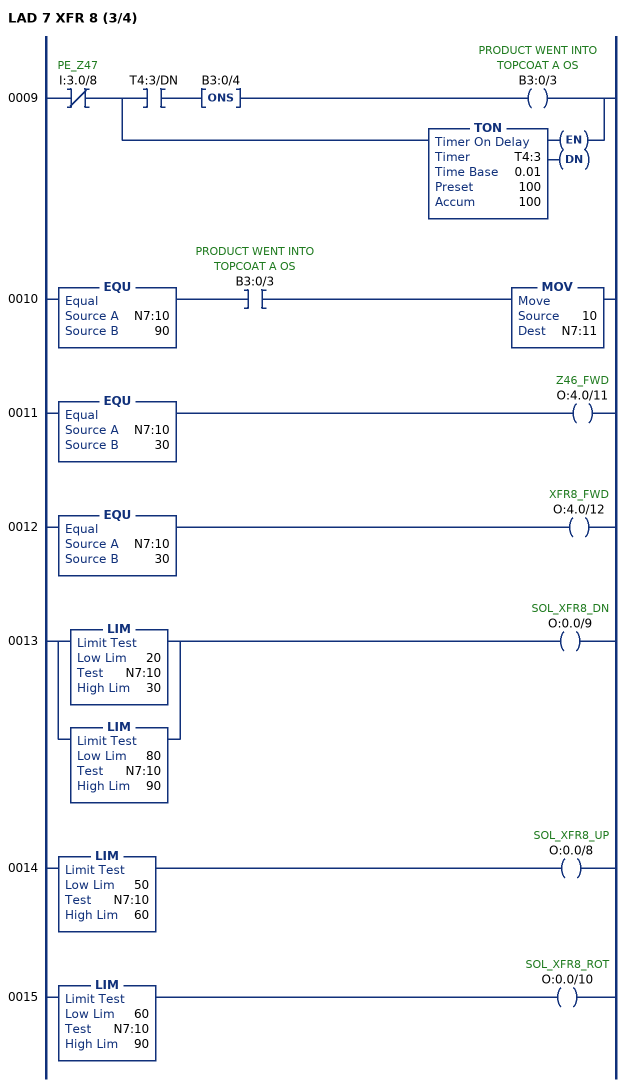
% Rung: 9 %
SOR XIO I:3.0/8 BST XIC T4:3/DN ONS B3:0/4 OTE B3:0/3 NXB TON T4:3 0.01 100 100 BND EOR
%   I:3.0/8  PE_Z47 %
%   B3:0/3  "PRODUCT WENT INTO TOPCOAT A OS" %
% Rung: 10 %
SOR EQU N7:10 90 XIC B3:0/3 MOV 10 N7:11 EOR
%   B3:0/3  "PRODUCT WENT INTO TOPCOAT A OS" %
% Rung: 11 %
SOR EQU N7:10 30 OTE O:4.0/11 EOR
%   O:4.0/11  Z46_FWD %
% Rung: 12 %
SOR EQU N7:10 30 OTE O:4.0/12 EOR
%   O:4.0/12  XFR8_FWD %
% Rung: 13 %
SOR BST LIM 20 N7:10 30 NXB LIM 80 N7:10 90 BND OTE O:0.0/9 EOR
%   O:0.0/9  SOL_XFR8_DN %
% Rung: 14 %
SOR LIM 50 N7:10 60 OTE O:0.0/8 EOR
%   O:0.0/8  SOL_XFR8_UP %
% Rung: 15 %
SOR LIM 60 N7:10 90 OTE O:0.0/10 EOR
%   O:0.0/10  SOL_XFR8_ROT %

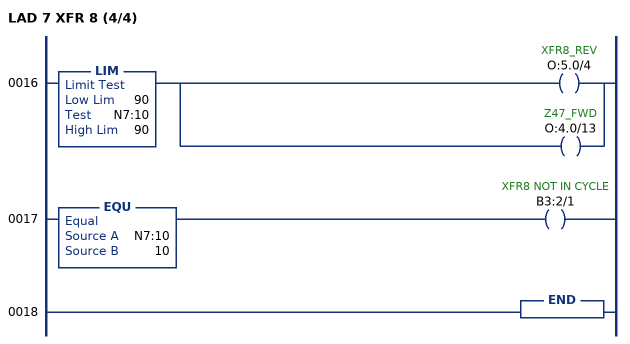
% Rung: 16 %
SOR LIM 90 N7:10 90 BST OTE O:5.0/4 NXB OTE O:4.0/13 BND EOR
%   O:5.0/4  XFR8_REV %
%   O:4.0/13  Z47_FWD %
% Rung: 17 %
SOR EQU N7:10 10 OTE B3:2/1 EOR
%   B3:2/1  "XFR8 NOT IN CYCLE" %
% Rung: 18 %
SOR END EOR

LADDER 8 "XFR 9"
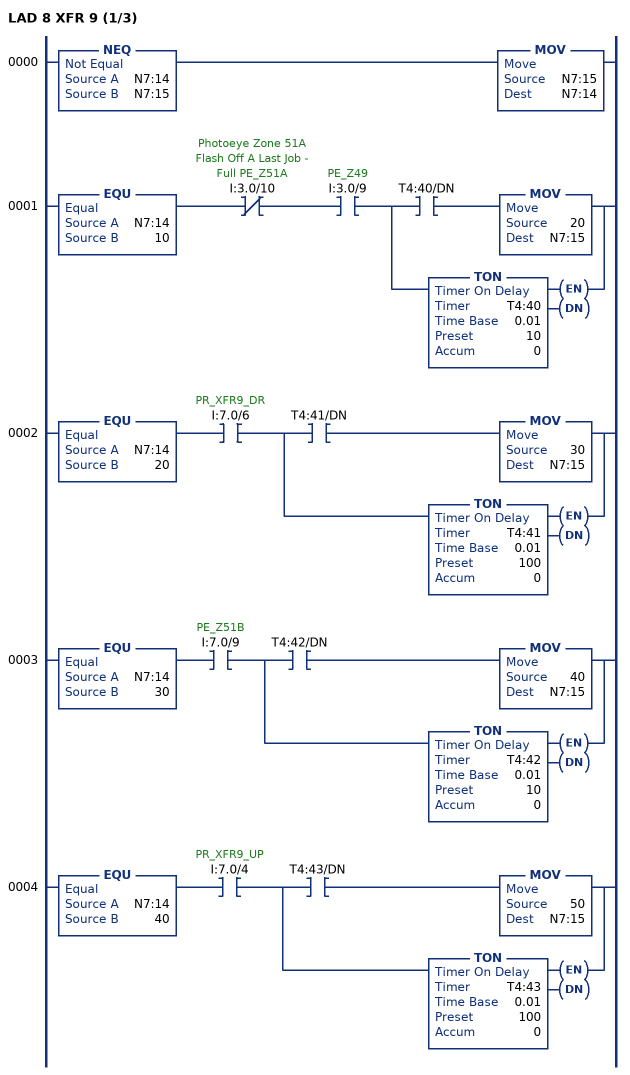
% Rung: 0 %
SOR NEQ N7:14 N7:15 MOV N7:15 N7:14 EOR
% Rung: 1 %
SOR EQU N7:14 10 XIO I:3.0/10 XIC I:3.0/9 BST XIC T4:40/DN MOV 20 N7:15 NXB TON T4:40 0.01 10 0 BND EOR
%   I:3.0/10  PE_Z51A  "Photoeye Zone 51A Flash Off A Last Job - Full" %
%   I:3.0/9  PE_Z49 %
% Rung: 2 %
SOR EQU N7:14 20 XIC I:7.0/6 BST XIC T4:41/DN MOV 30 N7:15 NXB TON T4:41 0.01 100 0 BND EOR
%   I:7.0/6  PR_XFR9_DR %
% Rung: 3 %
SOR EQU N7:14 30 XIC I:7.0/9 BST XIC T4:42/DN MOV 40 N7:15 NXB TON T4:42 0.01 10 0 BND EOR
%   I:7.0/9  PE_Z51B %
% Rung: 4 %
SOR EQU N7:14 40 XIC I:7.0/4 BST XIC T4:43/DN MOV 50 N7:15 NXB TON T4:43 0.01 100 0 BND EOR
%   I:7.0/4  PR_XFR9_UP %

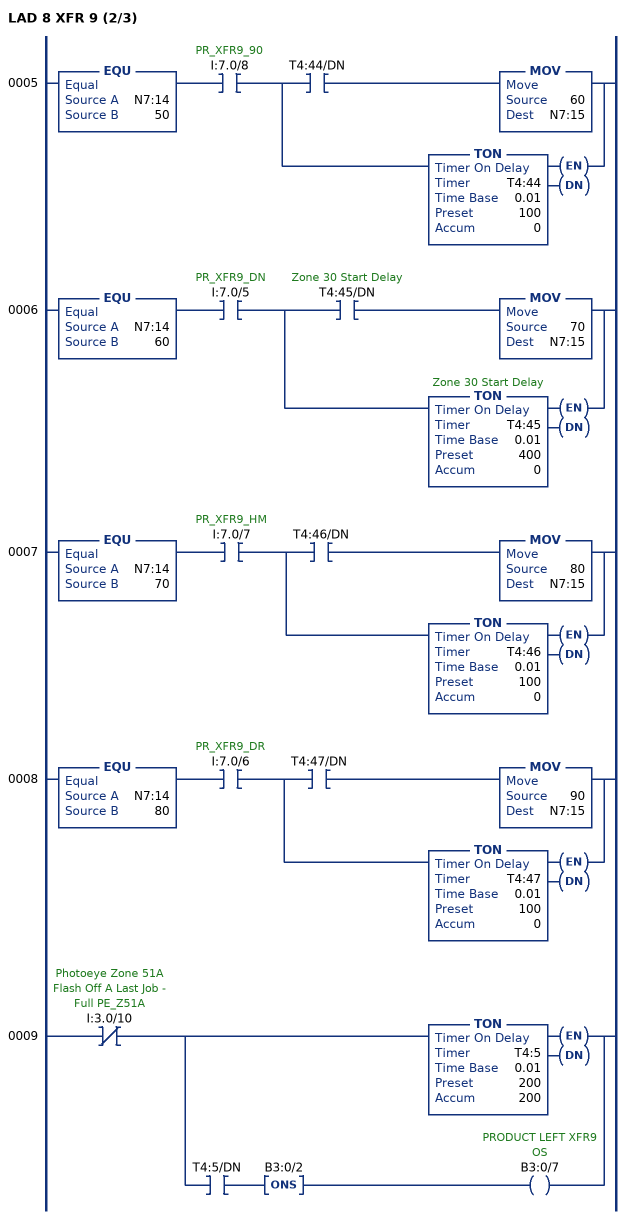
% Rung: 5 %
SOR EQU N7:14 50 XIC I:7.0/8 BST XIC T4:44/DN MOV 60 N7:15 NXB TON T4:44 0.01 100 0 BND EOR
%   I:7.0/8  PR_XFR9_90 %
% Rung: 6 %
SOR EQU N7:14 60 XIC I:7.0/5 BST XIC T4:45/DN MOV 70 N7:15 NXB TON T4:45 0.01 400 0 BND EOR
%   I:7.0/5  PR_XFR9_DN %
%   T4:45  "Zone 30 Start Delay" %
% Rung: 7 %
SOR EQU N7:14 70 XIC I:7.0/7 BST XIC T4:46/DN MOV 80 N7:15 NXB TON T4:46 0.01 100 0 BND EOR
%   I:7.0/7  PR_XFR9_HM %
% Rung: 8 %
SOR EQU N7:14 80 XIC I:7.0/6 BST XIC T4:47/DN MOV 90 N7:15 NXB TON T4:47 0.01 100 0 BND EOR
%   I:7.0/6  PR_XFR9_DR %
% Rung: 9 %
SOR XIO I:3.0/10 BST TON T4:5 0.01 200 200 NXB XIC T4:5/DN ONS B3:0/2 OTE B3:0/7 BND EOR
%   I:3.0/10  PE_Z51A  "Photoeye Zone 51A Flash Off A Last Job - Full" %
%   B3:0/7  "PRODUCT LEFT XFR9 OS" %

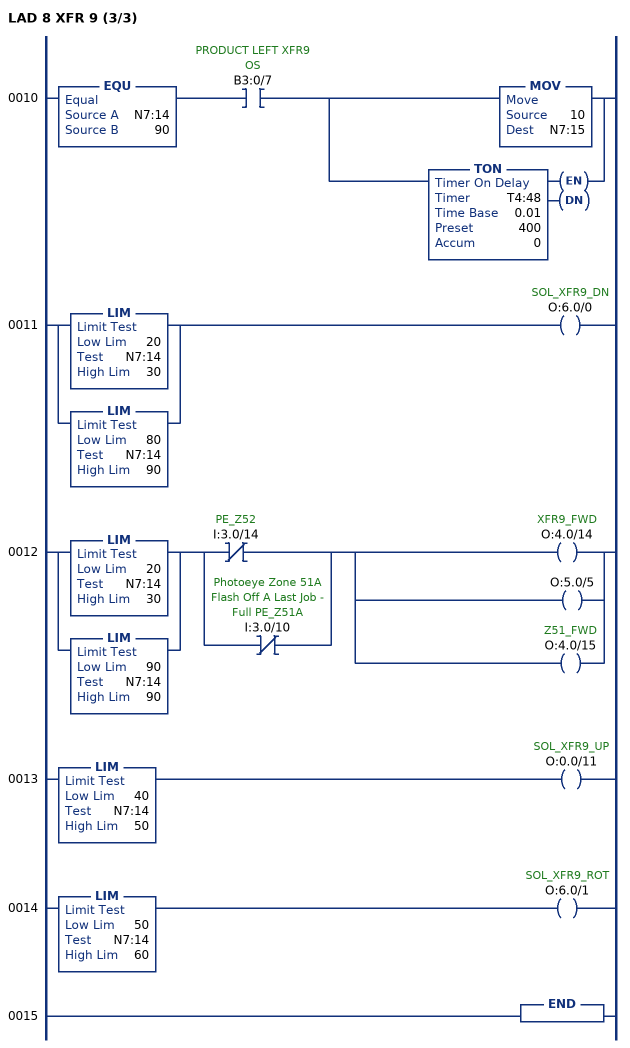
% Rung: 10 %
SOR EQU N7:14 90 XIC B3:0/7 BST MOV 10 N7:15 NXB TON T4:48 0.01 400 0 BND EOR
%   B3:0/7  "PRODUCT LEFT XFR9 OS" %
% Rung: 11 %
SOR BST LIM 20 N7:14 30 NXB LIM 80 N7:14 90 BND OTE O:6.0/0 EOR
%   O:6.0/0  SOL_XFR9_DN %
% Rung: 12 %
SOR BST LIM 20 N7:14 30 NXB LIM 90 N7:14 90 BND BST XIO I:3.0/14 NXB XIO I:3.0/10 BND BST OTE O:4.0/14 NXB OTE O:5.0/5 NXB OTE O:4.0/15 BND EOR
%   I:3.0/14  PE_Z52 %
%   I:3.0/10  PE_Z51A  "Photoeye Zone 51A Flash Off A Last Job - Full" %
%   O:4.0/14  XFR9_FWD %
%   O:4.0/15  Z51_FWD %
% Rung: 13 %
SOR LIM 40 N7:14 50 OTE O:0.0/11 EOR
%   O:0.0/11  SOL_XFR9_UP %
% Rung: 14 %
SOR LIM 50 N7:14 60 OTE O:6.0/1 EOR
%   O:6.0/1  SOL_XFR9_ROT %
% Rung: 15 %
SOR END EOR

LADDER 9 "XFR 10"
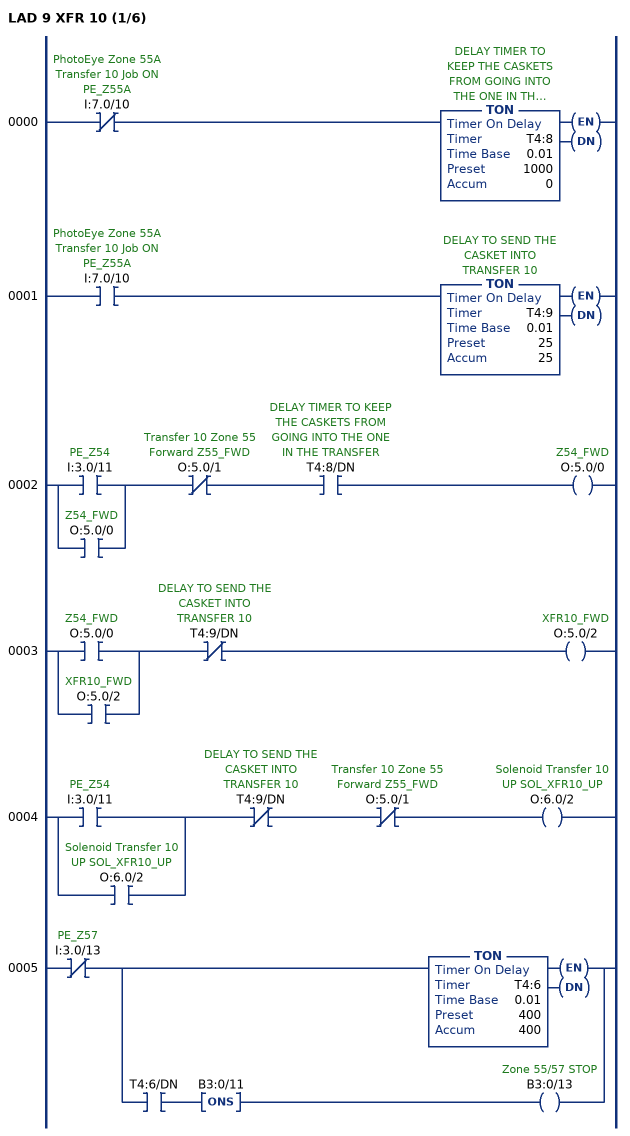
% Rung: 0 %
SOR XIO I:7.0/10 TON T4:8 0.01 1000 0 EOR
%   I:7.0/10  PE_Z55A  "PhotoEye Zone 55A Transfer 10 Job ON" %
%   T4:8  "DELAY TIMER TO KEEP THE CASKETS FROM GOING INTO THE ONE IN THE TRANSFER" %
% Rung: 1 %
SOR XIC I:7.0/10 TON T4:9 0.01 25 25 EOR
%   I:7.0/10  PE_Z55A  "PhotoEye Zone 55A Transfer 10 Job ON" %
%   T4:9  "DELAY TO SEND THE CASKET INTO TRANSFER 10" %
% Rung: 2 %
SOR BST XIC I:3.0/11 NXB XIC O:5.0/0 BND XIO O:5.0/1 XIC T4:8/DN OTE O:5.0/0 EOR
%   I:3.0/11  PE_Z54 %
%   O:5.0/0  Z54_FWD %
%   O:5.0/1  Z55_FWD  "Transfer 10 Zone 55 Forward" %
%   T4:8  "DELAY TIMER TO KEEP THE CASKETS FROM GOING INTO THE ONE IN THE TRANSFER" %
% Rung: 3 %
SOR BST XIC O:5.0/0 NXB XIC O:5.0/2 BND XIO T4:9/DN OTE O:5.0/2 EOR
%   O:5.0/0  Z54_FWD %
%   O:5.0/2  XFR10_FWD %
%   T4:9  "DELAY TO SEND THE CASKET INTO TRANSFER 10" %
% Rung: 4 %
SOR BST XIC I:3.0/11 NXB XIC O:6.0/2 BND XIO T4:9/DN XIO O:5.0/1 OTE O:6.0/2 EOR
%   I:3.0/11  PE_Z54 %
%   O:6.0/2  SOL_XFR10_UP  "Solenoid Transfer 10 UP" %
%   T4:9  "DELAY TO SEND THE CASKET INTO TRANSFER 10" %
%   O:5.0/1  Z55_FWD  "Transfer 10 Zone 55 Forward" %
% Rung: 5 %
SOR XIO I:3.0/13 BST TON T4:6 0.01 400 400 NXB XIC T4:6/DN ONS B3:0/11 OTE B3:0/13 BND EOR
%   I:3.0/13  PE_Z57 %
%   B3:0/13  "Zone 55/57 STOP" %

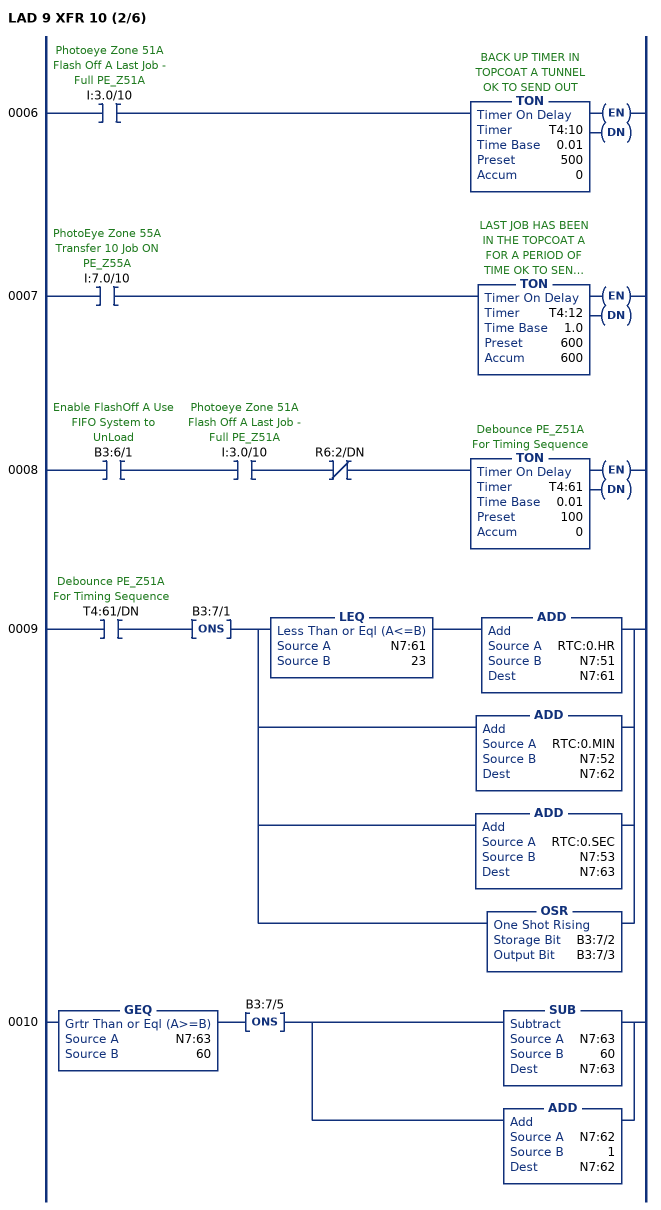
% Rung: 6 %
SOR XIC I:3.0/10 TON T4:10 0.01 500 0 EOR
%   I:3.0/10  PE_Z51A  "Photoeye Zone 51A Flash Off A Last Job - Full" %
%   T4:10  "BACK UP TIMER IN TOPCOAT A TUNNEL OK TO SEND OUT" %
% Rung: 7 %
SOR XIC I:7.0/10 TON T4:12 1.0 600 600 EOR
%   I:7.0/10  PE_Z55A  "PhotoEye Zone 55A Transfer 10 Job ON" %
%   T4:12  "LAST JOB HAS BEEN IN THE TOPCOAT A FOR A PERIOD OF TIME OK TO SEND OUT" %
% Rung: 8 %
SOR XIC B3:6/1 XIC I:3.0/10 XIO R6:2/DN TON T4:61 0.01 100 0 EOR
%   B3:6/1  "Enable FlashOff A Use FIFO System to UnLoad" %
%   I:3.0/10  PE_Z51A  "Photoeye Zone 51A Flash Off A Last Job - Full" %
%   T4:61  "Debounce PE_Z51A For Timing Sequence" %
% Rung: 9 %
SOR XIC T4:61/DN ONS B3:7/1 BST LEQ N7:61 23 ADD RTC:0.HR N7:51 N7:61 NXB ADD RTC:0.MIN N7:52 N7:62 NXB ADD RTC:0.SEC N7:53 N7:63 NXB OSR B3:7/2 B3:7/3 BND EOR
%   T4:61  "Debounce PE_Z51A For Timing Sequence" %
%   B3:7/3  "One Shot Rising FlashOff A Load Time into Stack" %
% Rung: 10 %
SOR GEQ N7:63 60 ONS B3:7/5 BST SUB N7:63 60 N7:63 NXB ADD N7:62 1 N7:62 BND EOR

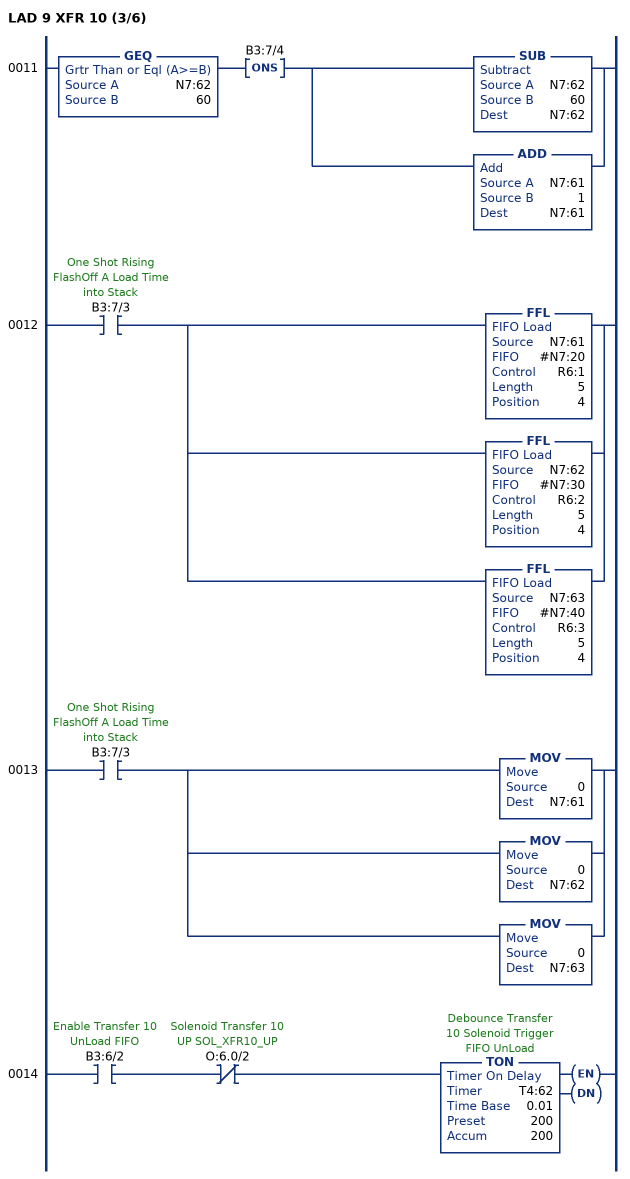
% Rung: 11 %
SOR GEQ N7:62 60 ONS B3:7/4 BST SUB N7:62 60 N7:62 NXB ADD N7:61 1 N7:61 BND EOR
% Rung: 12 %
SOR XIC B3:7/3 BST FFL N7:61 #N7:20 R6:1 5 4 NXB FFL N7:62 #N7:30 R6:2 5 4 NXB FFL N7:63 #N7:40 R6:3 5 4 BND EOR
%   B3:7/3  "One Shot Rising FlashOff A Load Time into Stack" %
% Rung: 13 %
SOR XIC B3:7/3 BST MOV 0 N7:61 NXB MOV 0 N7:62 NXB MOV 0 N7:63 BND EOR
%   B3:7/3  "One Shot Rising FlashOff A Load Time into Stack" %
% Rung: 14 %
SOR XIC B3:6/2 XIO O:6.0/2 TON T4:62 0.01 200 200 EOR
%   B3:6/2  "Enable Transfer 10 UnLoad FIFO" %
%   O:6.0/2  SOL_XFR10_UP  "Solenoid Transfer 10 UP" %
%   T4:62  "Debounce Transfer 10 Solenoid Trigger FIFO UnLoad" %

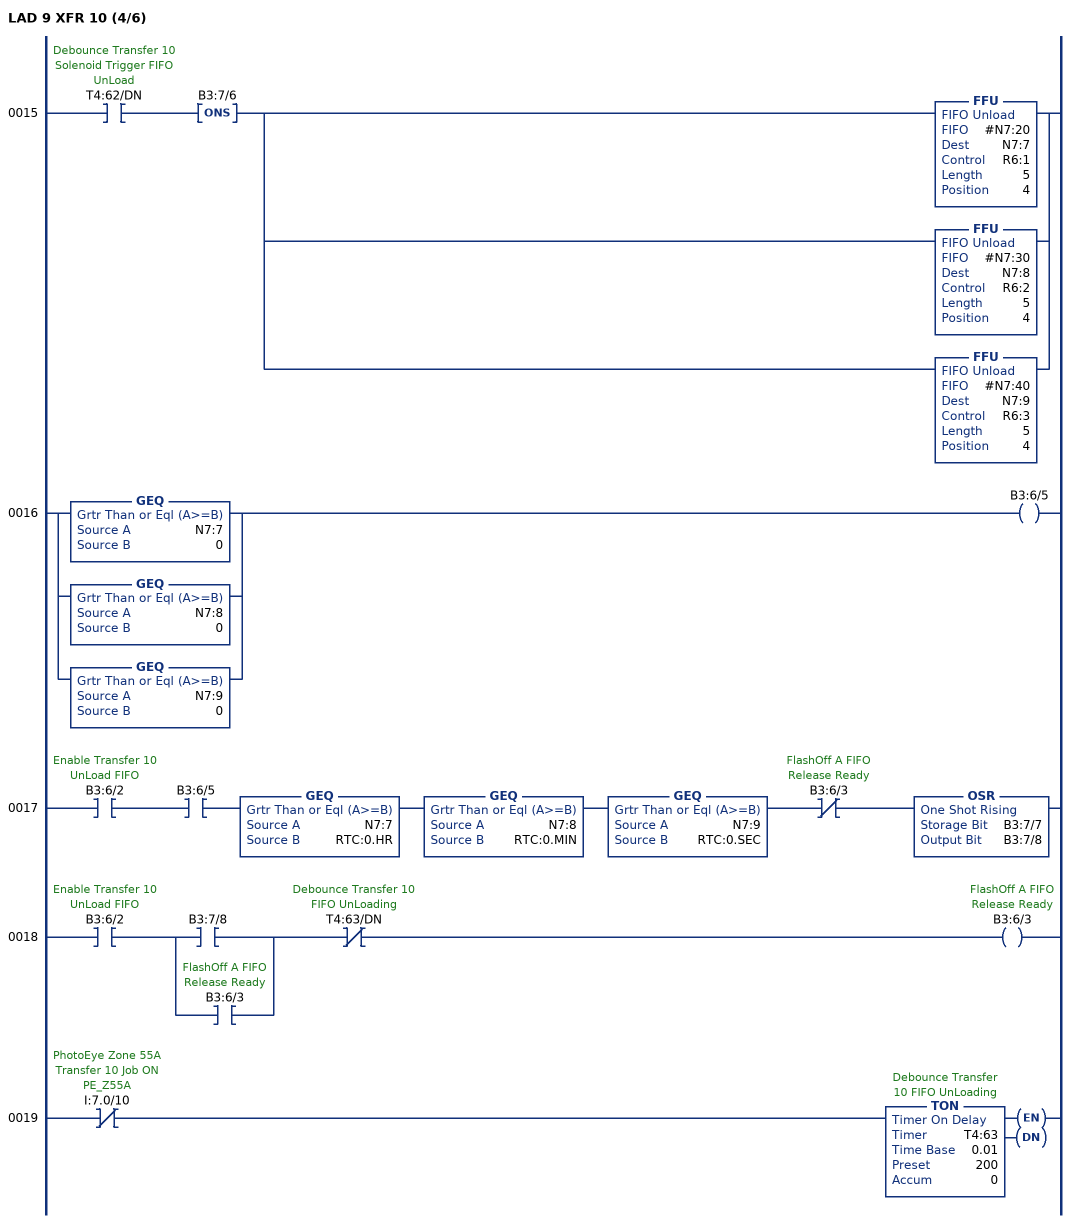
% Rung: 15 %
SOR XIC T4:62/DN ONS B3:7/6 BST FFU #N7:20 N7:7 R6:1 5 4 NXB FFU #N7:30 N7:8 R6:2 5 4 NXB FFU #N7:40 N7:9 R6:3 5 4 BND EOR
%   T4:62  "Debounce Transfer 10 Solenoid Trigger FIFO UnLoad" %
% Rung: 16 %
SOR BST GEQ N7:7 0 NXB GEQ N7:8 0 NXB GEQ N7:9 0 BND OTE B3:6/5 EOR
% Rung: 17 %
SOR XIC B3:6/2 XIC B3:6/5 GEQ N7:7 RTC:0.HR GEQ N7:8 RTC:0.MIN GEQ N7:9 RTC:0.SEC XIO B3:6/3 OSR B3:7/7 B3:7/8 EOR
%   B3:6/2  "Enable Transfer 10 UnLoad FIFO" %
%   B3:6/3  "FlashOff A FIFO Release Ready" %
% Rung: 18 %
SOR XIC B3:6/2 BST XIC B3:7/8 NXB XIC B3:6/3 BND XIO T4:63/DN OTE B3:6/3 EOR
%   B3:6/2  "Enable Transfer 10 UnLoad FIFO" %
%   B3:6/3  "FlashOff A FIFO Release Ready" %
%   T4:63  "Debounce Transfer 10 FIFO UnLoading" %
% Rung: 19 %
SOR XIO I:7.0/10 TON T4:63 0.01 200 0 EOR
%   I:7.0/10  PE_Z55A  "PhotoEye Zone 55A Transfer 10 Job ON" %
%   T4:63  "Debounce Transfer 10 FIFO UnLoading" %

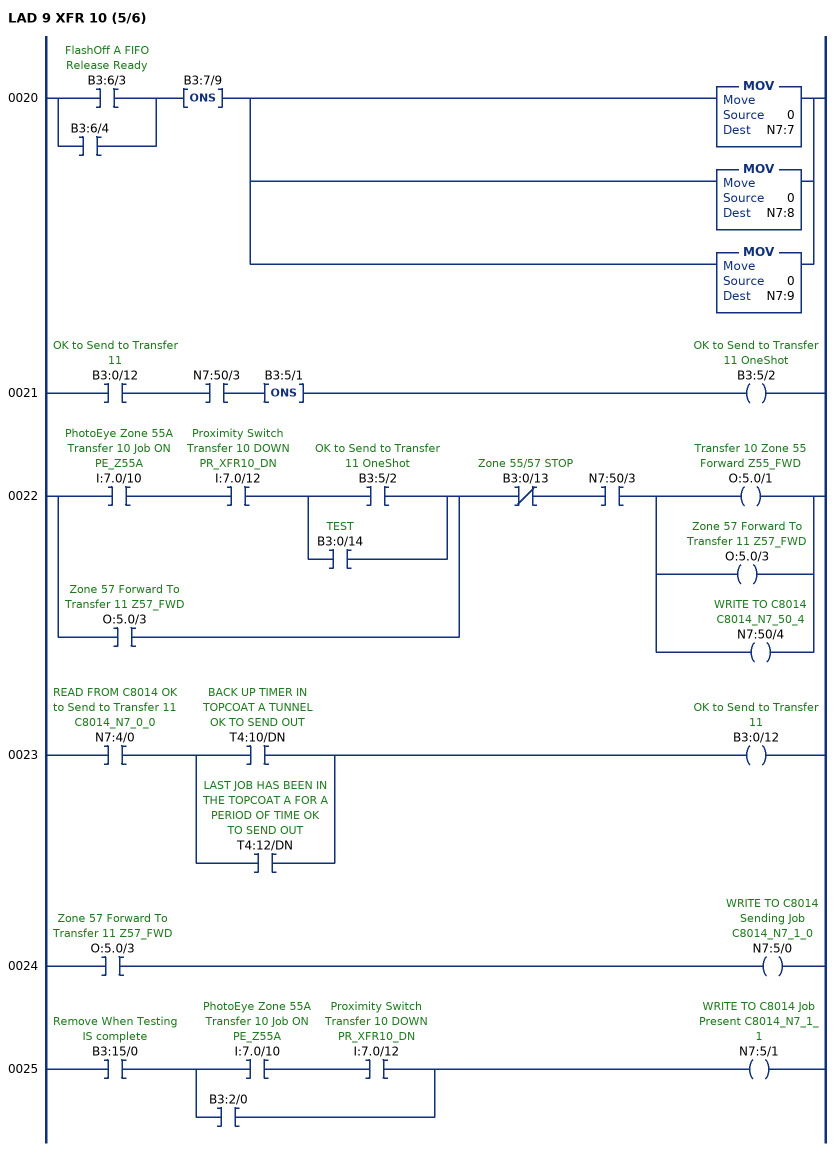
% Rung: 20 %
SOR BST XIC B3:6/3 NXB XIC B3:6/4 BND ONS B3:7/9 BST MOV 0 N7:7 NXB MOV 0 N7:8 NXB MOV 0 N7:9 BND EOR
%   B3:6/3  "FlashOff A FIFO Release Ready" %
% Rung: 21 %
SOR XIC B3:0/12 XIC N7:50/3 ONS B3:5/1 OTE B3:5/2 EOR
%   B3:0/12  "OK to Send to Transfer 11" %
%   B3:5/2  "OK to Send to Transfer 11 OneShot" %
% Rung: 22 %
SOR BST XIC I:7.0/10 XIC I:7.0/12 BST XIC B3:5/2 NXB XIC B3:0/14 BND NXB XIC O:5.0/3 BND XIO B3:0/13 XIC N7:50/3 BST OTE O:5.0/1 NXB OTE O:5.0/3 NXB OTE N7:50/4 BND EOR
%   I:7.0/10  PE_Z55A  "PhotoEye Zone 55A Transfer 10 Job ON" %
%   I:7.0/12  PR_XFR10_DN  "Proximity Switch Transfer 10 DOWN" %
%   B3:5/2  "OK to Send to Transfer 11 OneShot" %
%   B3:0/14  "TEST" %
%   O:5.0/3  Z57_FWD  "Zone 57 Forward To Transfer 11" %
%   B3:0/13  "Zone 55/57 STOP" %
%   O:5.0/1  Z55_FWD  "Transfer 10 Zone 55 Forward" %
%   N7:50/4  C8014_N7_50_4  "WRITE TO C8014" %
% Rung: 23 %
SOR XIC N7:4/0 BST XIC T4:10/DN NXB XIC T4:12/DN BND OTE B3:0/12 EOR
%   N7:4/0  C8014_N7_0_0  "READ FROM C8014 OK to Send to Transfer 11" %
%   T4:10  "BACK UP TIMER IN TOPCOAT A TUNNEL OK TO SEND OUT" %
%   T4:12  "LAST JOB HAS BEEN IN THE TOPCOAT A FOR A PERIOD OF TIME OK TO SEND OUT" %
%   B3:0/12  "OK to Send to Transfer 11" %
% Rung: 24 %
SOR XIC O:5.0/3 OTE N7:5/0 EOR
%   O:5.0/3  Z57_FWD  "Zone 57 Forward To Transfer 11" %
%   N7:5/0  C8014_N7_1_0  "WRITE TO C8014 Sending Job" %
% Rung: 25 %
SOR XIC B3:15/0 BST XIC I:7.0/10 XIC I:7.0/12 NXB XIC B3:2/0 BND OTE N7:5/1 EOR
%   B3:15/0  "Remove When Testing IS complete" %
%   I:7.0/10  PE_Z55A  "PhotoEye Zone 55A Transfer 10 Job ON" %
%   I:7.0/12  PR_XFR10_DN  "Proximity Switch Transfer 10 DOWN" %
%   N7:5/1  C8014_N7_1_1  "WRITE TO C8014 Job Present" %

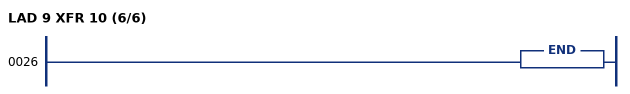
% Rung: 26 %
SOR END EOR

LADDER 10 "XFR 14"
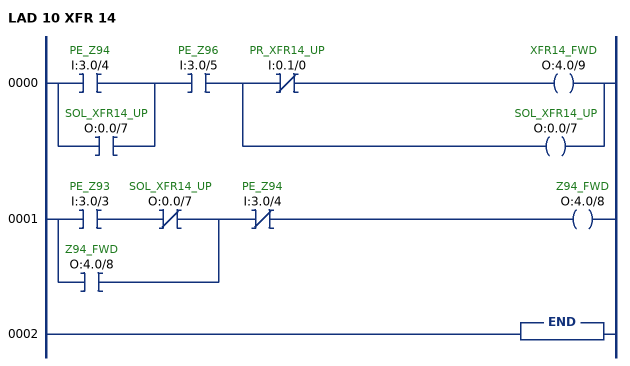
% Rung: 0 %
SOR BST XIC I:3.0/4 NXB XIC O:0.0/7 BND XIC I:3.0/5 BST XIO I:0.1/0 OTE O:4.0/9 NXB OTE O:0.0/7 BND EOR
%   I:3.0/4  PE_Z94 %
%   O:0.0/7  SOL_XFR14_UP %
%   I:3.0/5  PE_Z96 %
%   I:0.1/0  PR_XFR14_UP %
%   O:4.0/9  XFR14_FWD %
% Rung: 1 %
SOR BST XIC I:3.0/3 XIO O:0.0/7 NXB XIC O:4.0/8 BND XIO I:3.0/4 OTE O:4.0/8 EOR
%   I:3.0/3  PE_Z93 %
%   O:0.0/7  SOL_XFR14_UP %
%   O:4.0/8  Z94_FWD %
%   I:3.0/4  PE_Z94 %
% Rung: 2 %
SOR END EOR

LADDER 11 "RFID SB"
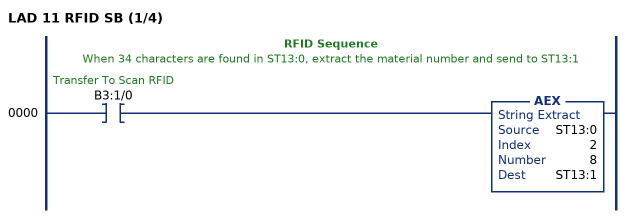
% Rung: 0 %
% TITLE: RFID Sequence %
% When 34 characters are found in ST13:0, extract the material number and send to ST13:1 %
SOR XIC B3:1/0 AEX ST13:0 2 8 ST13:1 EOR
%   B3:1/0  "Transfer To Scan RFID" %

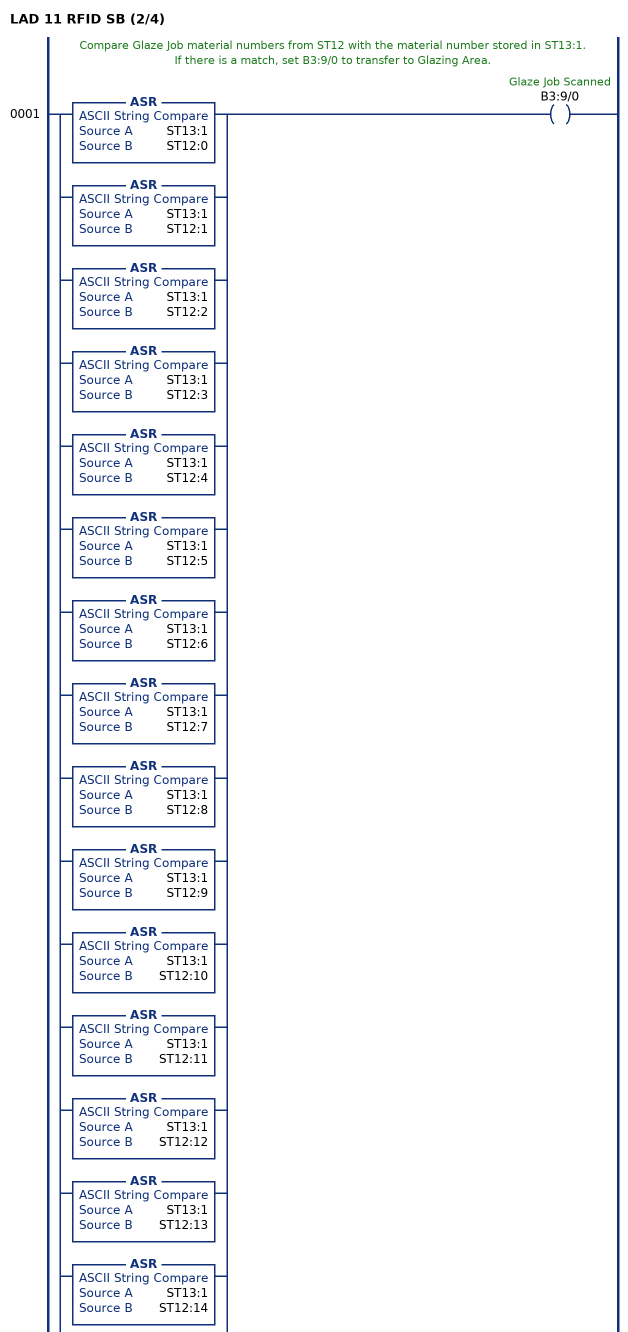

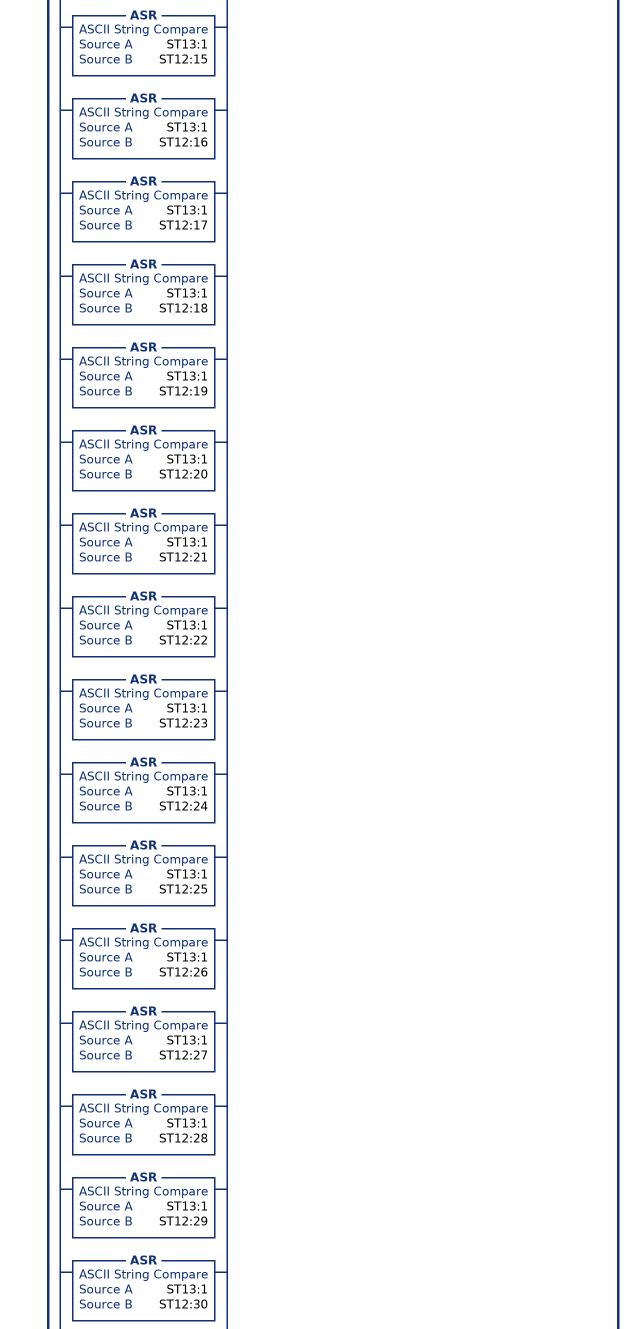

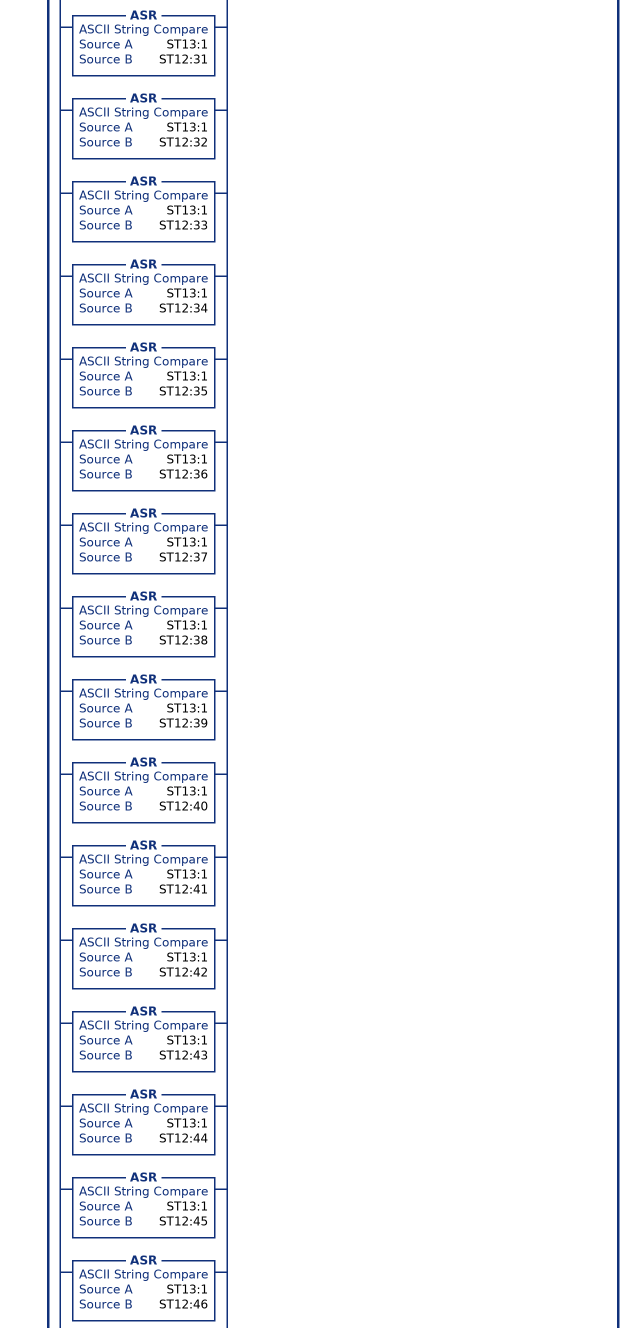

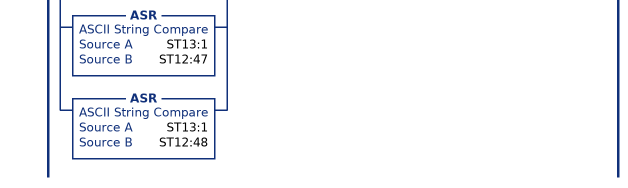
% Rung: 1 %
% Compare Glaze Job material numbers from ST12 with the material number stored in ST13:1. If there is a match, set B3:9/0 to transfer to Glazing Area. %
SOR BST ASR ST13:1 ST12:0 NXB ASR ST13:1 ST12:1 NXB ASR ST13:1 ST12:2 NXB ASR ST13:1 ST12:3 NXB ASR ST13:1 ST12:4 NXB ASR ST13:1 ST12:5 NXB ASR ST13:1 ST12:6 NXB ASR ST13:1 ST12:7 NXB ASR ST13:1 ST12:8 NXB ASR ST13:1 ST12:9 NXB ASR ST13:1 ST12:10 NXB ASR ST13:1 ST12:11 NXB ASR ST13:1 ST12:12 NXB ASR ST13:1 ST12:13 NXB ASR ST13:1 ST12:14 NXB ASR ST13:1 ST12:15 NXB ASR ST13:1 ST12:16 NXB ASR ST13:1 ST12:17 NXB ASR ST13:1 ST12:18 NXB ASR ST13:1 ST12:19 NXB ASR ST13:1 ST12:20 NXB ASR ST13:1 ST12:21 NXB ASR ST13:1 ST12:22 NXB ASR ST13:1 ST12:23 NXB ASR ST13:1 ST12:24 NXB ASR ST13:1 ST12:25 NXB ASR ST13:1 ST12:26 NXB ASR ST13:1 ST12:27 NXB ASR ST13:1 ST12:28 NXB ASR ST13:1 ST12:29 NXB ASR ST13:1 ST12:30 NXB ASR ST13:1 ST12:31 NXB ASR ST13:1 ST12:32 NXB ASR ST13:1 ST12:33 NXB ASR ST13:1 ST12:34 NXB ASR ST13:1 ST12:35 NXB ASR ST13:1 ST12:36 NXB ASR ST13:1 ST12:37 NXB ASR ST13:1 ST12:38 NXB ASR ST13:1 ST12:39 NXB ASR ST13:1 ST12:40 NXB ASR ST13:1 ST12:41 NXB ASR ST13:1 ST12:42 NXB ASR ST13:1 ST12:43 NXB ASR ST13:1 ST12:44 NXB ASR ST13:1 ST12:45 NXB ASR ST13:1 ST12:46 NXB ASR ST13:1 ST12:47 NXB ASR ST13:1 ST12:48 BND OTE B3:9/0 EOR
%   ST12:0  "Melrose Cherry" %
%   ST12:1  "Manchester Cherry IC" %
%   ST12:2  "Appalachian Cherry" %
%   ST12:3  "Chesapeake Cherry" %
%   ST12:4  "Virginia Rose Maple" %
%   ST12:5  "Dover Oak IC" %
%   ST12:6  "Woodstock Oak IC" %
%   ST12:7  "Akron Oak" %
%   ST12:8  "Magnolia" %
%   ST12:9  "Magnolia" %
%   ST12:10  "Lincoln" %
%   ST12:11  "Marion" %
%   ST12:12  "Coventry" %
%   ST12:13  "Dakota" %
%   ST12:14  "23rd Psalm" %
%   ST12:15  "Washington" %
%   ST12:16  "Sequoia Pilgrim" %
%   ST12:17  "Sebring" %
%   ST12:18  "Sebring" %
%   ST12:19  "Dayton" %
%   ST12:20  "Sandy Birch" %
%   ST12:21  "Sandy Birch" %
%   ST12:22  "Sandy Birch" %
%   ST12:23  "Fractional Unit" %
%   ST12:24  "Fractional Unit" %
%   ST12:25  "Fractional Unit" %
%   ST12:26  "Fractional Unit" %
%   ST12:27  "Fractional Unit" %
%   ST12:28  "Fractional Unit" %
%   ST12:29  "Fractional Unit" %
%   ST12:30  "Fractional Unit" %
%   ST12:31  "Fractional Unit" %
%   ST12:32  "Fractional Unit" %
%   ST12:33  "Fractional Unit" %
%   ST12:34  "Fractional Unit" %
%   ST12:35  "Fractional Unit" %
%   ST12:36  "Fractional Unit" %
%   ST12:37  "Fractional Unit" %
%   ST12:38  "Fractional Unit" %
%   ST12:39  "Fractional Unit" %
%   ST12:40  "Fractional Unit" %
%   ST12:41  "Fractional Unit" %
%   ST12:42  "Fractional Unit" %
%   ST12:44  "Dakota" %
%   ST12:47  "Dakota" %
%   B3:9/0  "Glaze Job Scanned" %

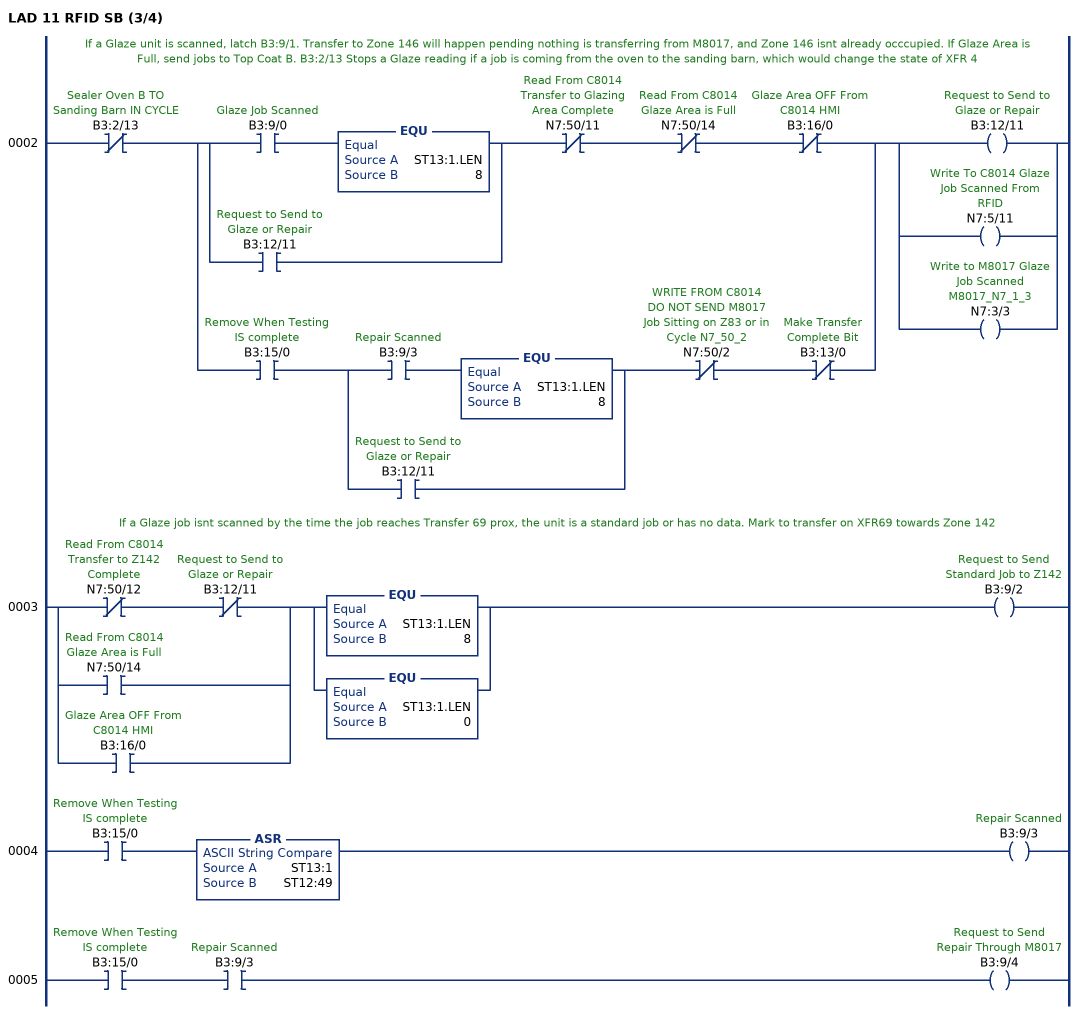
% Rung: 2 %
% If a Glaze unit is scanned, latch B3:9/1. Transfer to Zone 146 will happen pending nothing is transferring from M8017, and Zone 146 isnt already occcupied. If Glaze Area is Full, send jobs to Top Coat B. B3:2/13 Stops a Glaze reading if a job is coming from the oven to the sanding barn, which would change the state of XFR 4 %
SOR XIO B3:2/13 BST BST XIC B3:9/0 EQU ST13:1.LEN 8 NXB XIC B3:12/11 BND XIO N7:50/11 XIO N7:50/14 XIO B3:16/0 NXB XIC B3:15/0 BST XIC B3:9/3 EQU ST13:1.LEN 8 NXB XIC B3:12/11 BND XIO N7:50/2 XIO B3:13/0 BND BST OTE B3:12/11 NXB OTE N7:5/11 NXB OTE N7:3/3 BND EOR
%   B3:2/13  "Sealer Oven B TO Sanding Barn IN CYCLE" %
%   B3:9/0  "Glaze Job Scanned" %
%   B3:12/11  "Request to Send to Glaze or Repair" %
%   N7:50/11  "Read From C8014 Transfer to Glazing Area Complete" %
%   N7:50/14  "Read From C8014 Glaze Area is Full" %
%   B3:16/0  "Glaze Area OFF From C8014 HMI" %
%   B3:15/0  "Remove When Testing IS complete" %
%   B3:9/3  "Repair Scanned" %
%   N7:50/2  N7_50_2  "WRITE FROM C8014 DO NOT SEND M8017 Job Sitting on Z83 or in Cycle" %
%   B3:13/0  "Make Transfer Complete Bit" %
%   N7:5/11  "Write To C8014 Glaze Job Scanned From RFID" %
%   N7:3/3  M8017_N7_1_3  "Write to M8017 Glaze Job Scanned" %
% Rung: 3 %
% If a Glaze job isnt scanned by the time the job reaches Transfer 69 prox, the unit is a standard job or has no data. Mark to transfer on XFR69 towards Zone 142 %
SOR BST XIO N7:50/12 XIO B3:12/11 NXB XIC N7:50/14 NXB XIC B3:16/0 BND BST EQU ST13:1.LEN 8 NXB EQU ST13:1.LEN 0 BND OTE B3:9/2 EOR
%   N7:50/12  "Read From C8014 Transfer to Z142 Complete" %
%   B3:12/11  "Request to Send to Glaze or Repair" %
%   N7:50/14  "Read From C8014 Glaze Area is Full" %
%   B3:16/0  "Glaze Area OFF From C8014 HMI" %
%   B3:9/2  "Request to Send Standard Job to Z142" %
% Rung: 4 %
SOR XIC B3:15/0 ASR ST13:1 ST12:49 OTE B3:9/3 EOR
%   B3:15/0  "Remove When Testing IS complete" %
%   B3:9/3  "Repair Scanned" %
% Rung: 5 %
SOR XIC B3:15/0 XIC B3:9/3 OTE B3:9/4 EOR
%   B3:15/0  "Remove When Testing IS complete" %
%   B3:9/3  "Repair Scanned" %
%   B3:9/4  "Request to Send Repair Through M8017" %

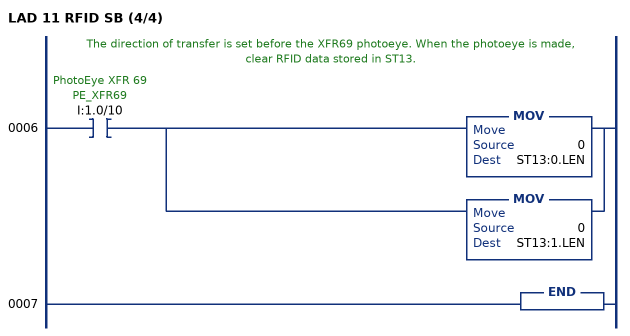
% Rung: 6 %
% The direction of transfer is set before the XFR69 photoeye. When the photoeye is made, clear RFID data stored in ST13. %
SOR XIC I:1.0/10 BST MOV 0 ST13:0.LEN NXB MOV 0 ST13:1.LEN BND EOR
%   I:1.0/10  PE_XFR69  "PhotoEye XFR 69" %
% Rung: 7 %
SOR END EOR

LADDER 12 "Z24_Z21"
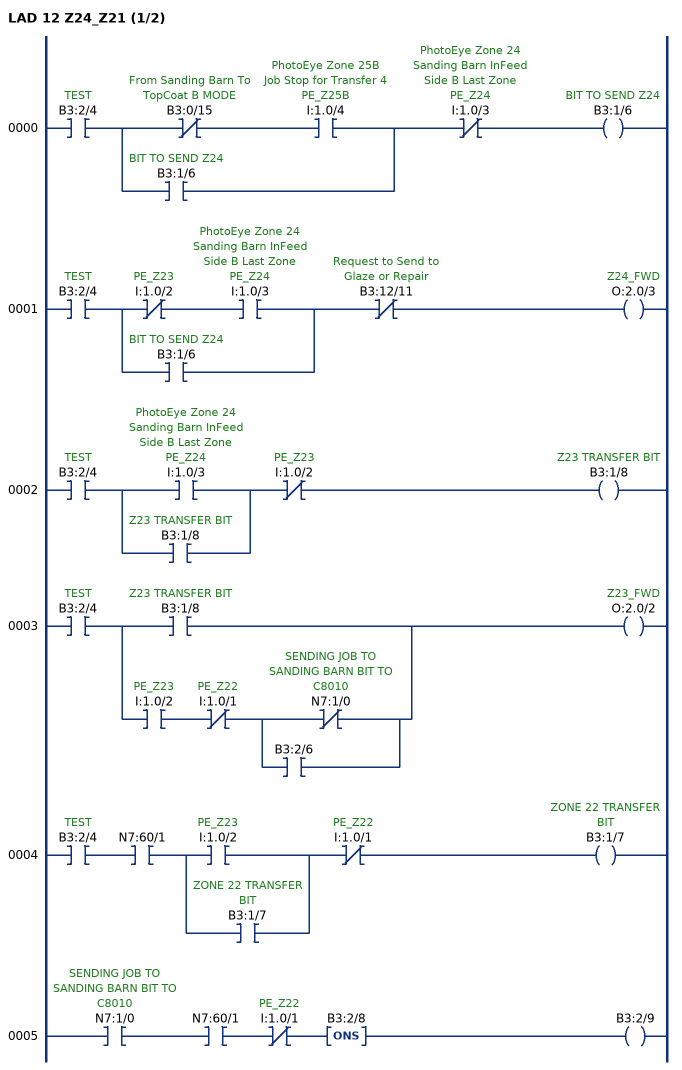
% Rung: 0 %
SOR XIC B3:2/4 BST XIO B3:0/15 XIC I:1.0/4 NXB XIC B3:1/6 BND XIO I:1.0/3 OTE B3:1/6 EOR
%   B3:2/4  "TEST" %
%   B3:0/15  "From Sanding Barn To TopCoat B MODE" %
%   I:1.0/4  PE_Z25B  "PhotoEye Zone 25B Job Stop for Transfer 4" %
%   B3:1/6  "BIT TO SEND Z24" %
%   I:1.0/3  PE_Z24  "PhotoEye Zone 24 Sanding Barn InFeed Side B Last Zone" %
% Rung: 1 %
SOR XIC B3:2/4 BST XIO I:1.0/2 XIC I:1.0/3 NXB XIC B3:1/6 BND XIO B3:12/11 OTE O:2.0/3 EOR
%   B3:2/4  "TEST" %
%   I:1.0/2  PE_Z23 %
%   I:1.0/3  PE_Z24  "PhotoEye Zone 24 Sanding Barn InFeed Side B Last Zone" %
%   B3:1/6  "BIT TO SEND Z24" %
%   B3:12/11  "Request to Send to Glaze or Repair" %
%   O:2.0/3  Z24_FWD %
% Rung: 2 %
SOR XIC B3:2/4 BST XIC I:1.0/3 NXB XIC B3:1/8 BND XIO I:1.0/2 OTE B3:1/8 EOR
%   B3:2/4  "TEST" %
%   I:1.0/3  PE_Z24  "PhotoEye Zone 24 Sanding Barn InFeed Side B Last Zone" %
%   B3:1/8  "Z23 TRANSFER BIT" %
%   I:1.0/2  PE_Z23 %
% Rung: 3 %
SOR XIC B3:2/4 BST XIC B3:1/8 NXB XIC I:1.0/2 XIO I:1.0/1 BST XIO N7:1/0 NXB XIC B3:2/6 BND BND OTE O:2.0/2 EOR
%   B3:2/4  "TEST" %
%   B3:1/8  "Z23 TRANSFER BIT" %
%   I:1.0/2  PE_Z23 %
%   I:1.0/1  PE_Z22 %
%   N7:1/0  "SENDING JOB TO SANDING BARN BIT TO C8010" %
%   O:2.0/2  Z23_FWD %
% Rung: 4 %
SOR XIC B3:2/4 XIC N7:60/1 BST XIC I:1.0/2 NXB XIC B3:1/7 BND XIO I:1.0/1 OTE B3:1/7 EOR
%   B3:2/4  "TEST" %
%   I:1.0/2  PE_Z23 %
%   B3:1/7  "ZONE 22 TRANSFER BIT" %
%   I:1.0/1  PE_Z22 %
% Rung: 5 %
SOR XIC N7:1/0 XIC N7:60/1 XIO I:1.0/1 ONS B3:2/8 OTE B3:2/9 EOR
%   N7:1/0  "SENDING JOB TO SANDING BARN BIT TO C8010" %
%   I:1.0/1  PE_Z22 %

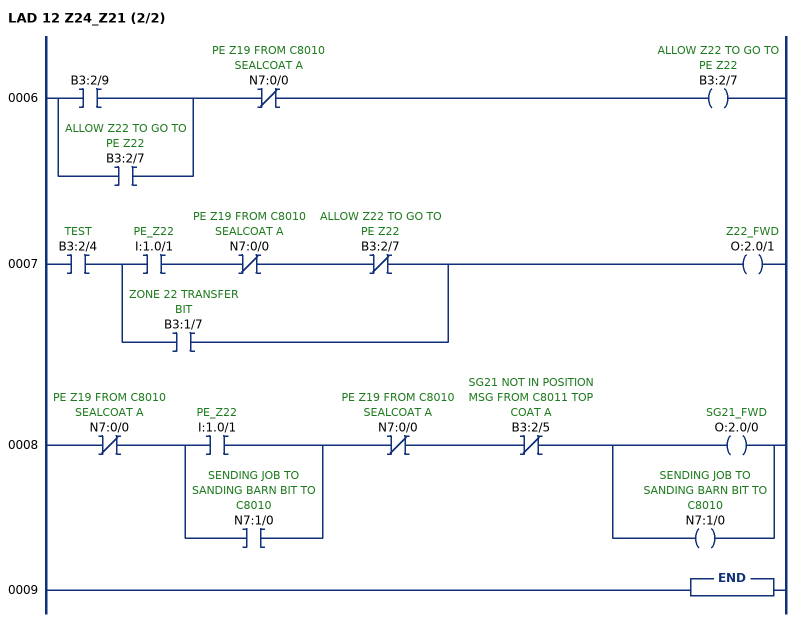
% Rung: 6 %
SOR BST XIC B3:2/9 NXB XIC B3:2/7 BND XIO N7:0/0 OTE B3:2/7 EOR
%   B3:2/7  "ALLOW Z22 TO GO TO PE Z22" %
%   N7:0/0  "PE Z19 FROM C8010 SEALCOAT A" %
% Rung: 7 %
SOR XIC B3:2/4 BST XIC I:1.0/1 XIO N7:0/0 XIO B3:2/7 NXB XIC B3:1/7 BND OTE O:2.0/1 EOR
%   B3:2/4  "TEST" %
%   I:1.0/1  PE_Z22 %
%   N7:0/0  "PE Z19 FROM C8010 SEALCOAT A" %
%   B3:2/7  "ALLOW Z22 TO GO TO PE Z22" %
%   B3:1/7  "ZONE 22 TRANSFER BIT" %
%   O:2.0/1  Z22_FWD %
% Rung: 8 %
SOR XIO N7:0/0 BST XIC I:1.0/1 NXB XIC N7:1/0 BND XIO N7:0/0 XIO B3:2/5 BST OTE O:2.0/0 NXB OTE N7:1/0 BND EOR
%   N7:0/0  "PE Z19 FROM C8010 SEALCOAT A" %
%   I:1.0/1  PE_Z22 %
%   N7:1/0  "SENDING JOB TO SANDING BARN BIT TO C8010" %
%   B3:2/5  "SG21 NOT IN POSITION MSG FROM C8011 TOP COAT A" %
%   O:2.0/0  SG21_FWD %
% Rung: 9 %
SOR END EOR

LADDER 13 "Z90_Z92"
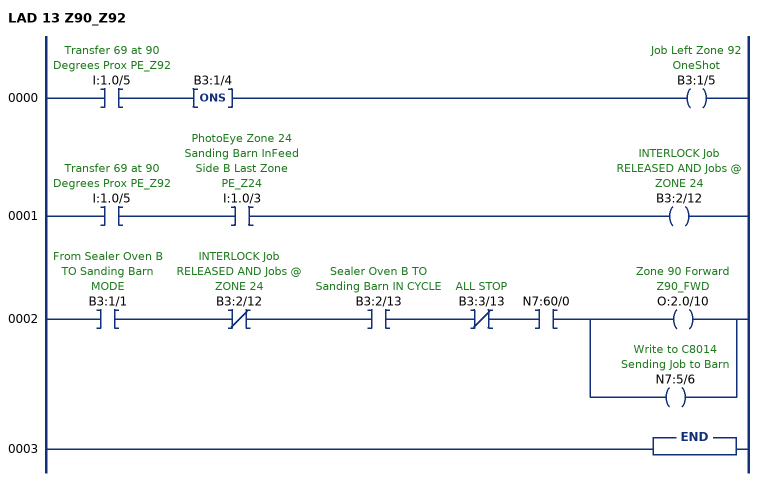
% Rung: 0 %
SOR XIC I:1.0/5 ONS B3:1/4 OTE B3:1/5 EOR
%   I:1.0/5  PE_Z92  "Transfer 69 at 90 Degrees Prox" %
%   B3:1/5  "Job Left Zone 92 OneShot" %
% Rung: 1 %
SOR XIC I:1.0/5 XIC I:1.0/3 OTE B3:2/12 EOR
%   I:1.0/5  PE_Z92  "Transfer 69 at 90 Degrees Prox" %
%   I:1.0/3  PE_Z24  "PhotoEye Zone 24 Sanding Barn InFeed Side B Last Zone" %
%   B3:2/12  "INTERLOCK Job RELEASED AND Jobs @ ZONE 24" %
% Rung: 2 %
SOR XIC B3:1/1 XIO B3:2/12 XIC B3:2/13 XIO B3:3/13 XIC N7:60/0 BST OTE O:2.0/10 NXB OTE N7:5/6 BND EOR
%   B3:1/1  "From Sealer Oven B TO Sanding Barn MODE" %
%   B3:2/12  "INTERLOCK Job RELEASED AND Jobs @ ZONE 24" %
%   B3:2/13  "Sealer Oven B TO Sanding Barn IN CYCLE" %
%   B3:3/13  "ALL STOP" %
%   O:2.0/10  Z90_FWD  "Zone 90 Forward" %
%   N7:5/6  "Write to C8014 Sending Job to Barn" %
% Rung: 3 %
SOR END EOR

LADDER 15 "COMM"
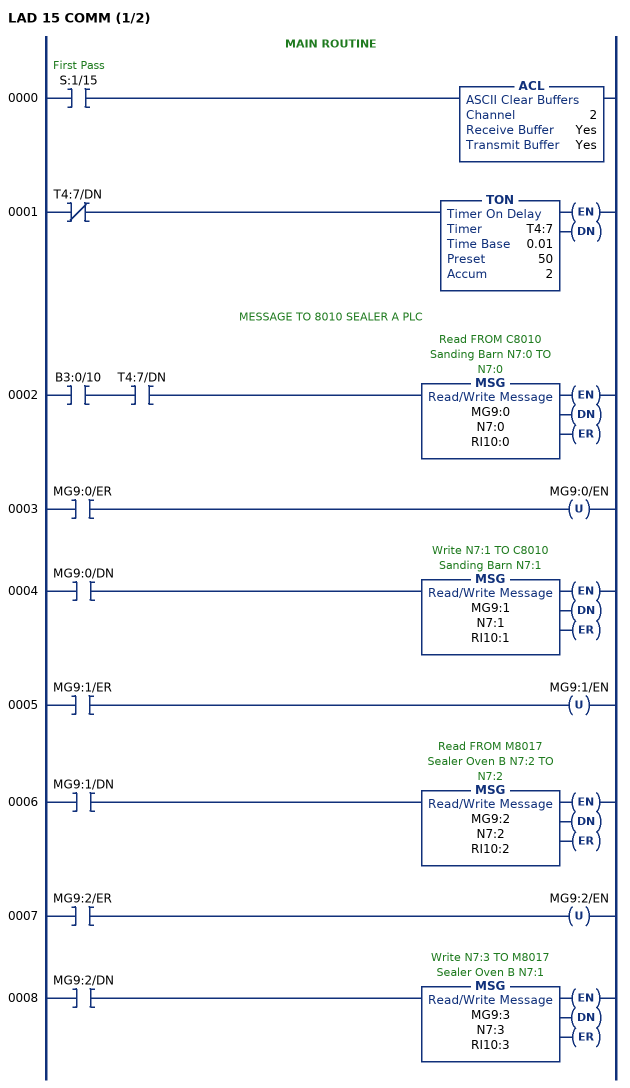
% Rung: 0 %
% TITLE: MAIN ROUTINE %
SOR XIC S:1/15 ACL 2 Yes Yes EOR
%   S:1/15  "First Pass" %
% Rung: 1 %
SOR XIO T4:7/DN TON T4:7 0.01 50 2 EOR
% Rung: 2 %
% MESSAGE TO 8010 SEALER A PLC %
SOR XIC B3:0/10 XIC T4:7/DN MSG MG9:0 N7:0 RI10:0 EOR
%   MSG set-up: 500CPU Read | 33 | 1 | N7:0 | N7:0 | 0 | 0 | 0 | 172.18.35.30 | 0 | 0 | 172.18.35.30 | RI10:0 %
%   MG9:0  "Read FROM C8010 Sanding Barn N7:0 TO N7:0" %
%   N7:0  "FROM SEALER A" %
% Rung: 3 %
SOR XIC MG9:0/ER OTU MG9:0/EN EOR
% Rung: 4 %
SOR XIC MG9:0/DN MSG MG9:1 N7:1 RI10:1 EOR
%   MSG set-up: 500CPU Write | 33 | 1 | N7:1 | N7:1 | 0 | 0 | 0 | 172.18.35.30 | 0 | 0 | 172.18.35.30 | RI10:1 %
%   MG9:1  "Write N7:1 TO C8010 Sanding Barn N7:1" %
%   N7:1  WRITE_TO_SEALER %
% Rung: 5 %
SOR XIC MG9:1/ER OTU MG9:1/EN EOR
% Rung: 6 %
SOR XIC MG9:1/DN MSG MG9:2 N7:2 RI10:2 EOR
%   MSG set-up: 500CPU Read | 33 | 1 | N7:0 | N7:2 | 0 | 0 | 0 | 172.18.35.39 | 0 | 0 | 172.18.35.39 | RI10:2 %
%   MG9:2  "Read FROM M8017 Sealer Oven B N7:2 TO N7:2" %
%   N7:2  "FROM_M8017_OVEN_2" %
% Rung: 7 %
SOR XIC MG9:2/ER OTU MG9:2/EN EOR
% Rung: 8 %
SOR XIC MG9:2/DN MSG MG9:3 N7:3 RI10:3 EOR
%   MSG set-up: 500CPU Write | 33 | 1 | N7:1 | N7:3 | 0 | 0 | 0 | 172.18.35.39 | 0 | 0 | 172.18.35.39 | RI10:3 %
%   MG9:3  "Write N7:3 TO M8017 Sealer Oven B N7:1" %
%   N7:3  "WRITE TO OVEN" %

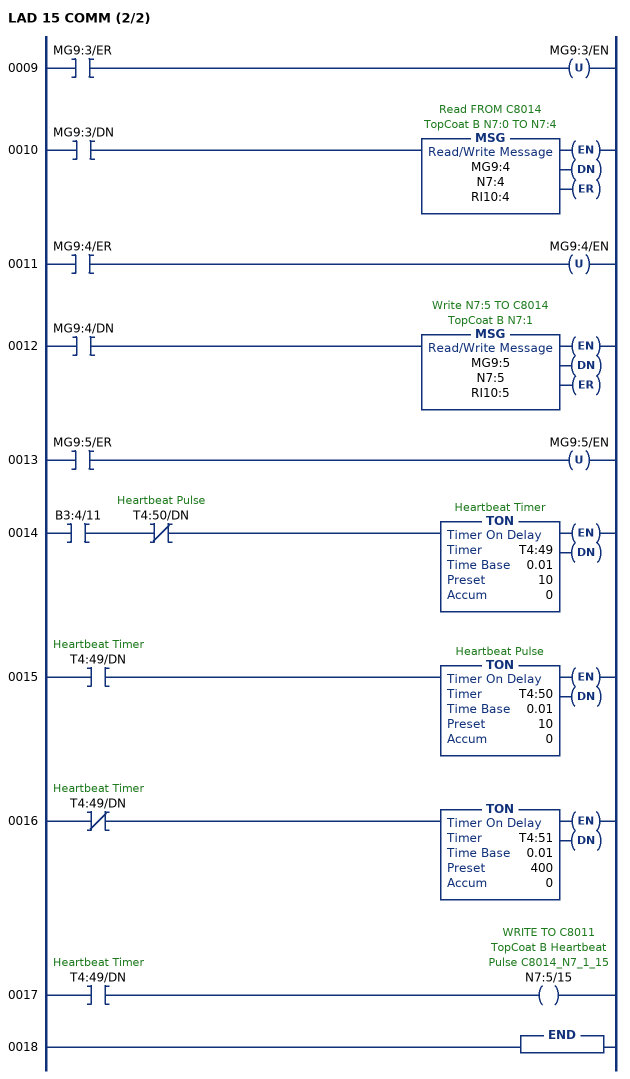
% Rung: 9 %
SOR XIC MG9:3/ER OTU MG9:3/EN EOR
% Rung: 10 %
SOR XIC MG9:3/DN MSG MG9:4 N7:4 RI10:4 EOR
%   MSG set-up: 500CPU Read | 33 | 1 | N7:0 | N7:4 | 0 | 0 | 0 | 172.18.35.19 | 0 | 0 | 172.18.35.19 | RI10:4 %
%   MG9:4  "Read FROM C8014 TopCoat B N7:0 TO N7:4" %
%   N7:4  READ_FROM_TOPCOAT_B %
% Rung: 11 %
SOR XIC MG9:4/ER OTU MG9:4/EN EOR
% Rung: 12 %
SOR XIC MG9:4/DN MSG MG9:5 N7:5 RI10:5 EOR
%   MSG set-up: 500CPU Write | 33 | 1 | N7:1 | N7:5 | 0 | 0 | 0 | 172.18.35.19 | 0 | 0 | 172.18.35.19 | RI10:5 %
%   MG9:5  "Write N7:5 TO C8014 TopCoat B N7:1" %
%   N7:5  WRITE_TO_TOPCOAT_B %
% Rung: 13 %
SOR XIC MG9:5/ER OTU MG9:5/EN EOR
% Rung: 14 %
SOR XIC B3:4/11 XIO T4:50/DN TON T4:49 0.01 10 0 EOR
%   T4:50  "Heartbeat Pulse" %
%   T4:49  "Heartbeat Timer" %
% Rung: 15 %
SOR XIC T4:49/DN TON T4:50 0.01 10 0 EOR
%   T4:49  "Heartbeat Timer" %
%   T4:50  "Heartbeat Pulse" %
% Rung: 16 %
SOR XIO T4:49/DN TON T4:51 0.01 400 0 EOR
%   T4:49  "Heartbeat Timer" %
% Rung: 17 %
SOR XIC T4:49/DN OTE N7:5/15 EOR
%   T4:49  "Heartbeat Timer" %
%   N7:5/15  C8014_N7_1_15  "WRITE TO C8011 TopCoat B Heartbeat Pulse" %
% Rung: 18 %
SOR END EOR

LADDER 16 "XFR 69"
